// TwinCAT 3 PLC project PLCStudent
// ProgramVersion: 3.1.4022.4
// libraries:
//   Tc2_Standard, * (Beckhoff Automation GmbH)
//   Tc2_System, * (Beckhoff Automation GmbH)
//   Tc3_Module, * (Beckhoff Automation GmbH)
//   VisuSymbols,3.5.10.0,System
// project tree:
//   / GlobalTextList.TcGTLO, PlcTask.TcTTO (not stored), Visualization Manager.TcVMO (not stored)
//   GVLs/ GVL.TcGVL
//   POUs/ Control_AGV_SFC.TcPOU, Display_Pos.TcPOU, MAIN.TcPOU
//   VISUs/ Control_HMI.TcVIS
// (motion and I/O tree: see PLC project plcsim)
// real-time tasks:
//   TASK PlcTask: cycle T#20ms, priority 20, ADS port 350
// variable links:
//   PLCSim/PLCSim Instance <-> PLCStudent/PLCStudent Instance
//     PlcTask Inputs/GVL.iiGotoPos <-> PlcTask Outputs/GVL.qiGotoPos
//     PlcTask Inputs/GVL.ixPLCStrobe <-> PlcTask Outputs/GVL.qxPLCStrobe
//     PlcTask Outputs/GVL.qiAtPos <-> PlcTask Inputs/GVL.iiAtPos
//     PlcTask Outputs/GVL.qxAGVStrobe <-> PlcTask Inputs/GVL.ixAGVStrobe

// ---- GVLs/GVL.TcGVL
{attribute 'qualified_only'}
VAR_GLOBAL
//Input to PLC from process
	ixAGVStrobe		AT %I*:	BOOL;	(* AGV strobe signal *)
	iiAtPos			AT %I*:	INT;	(* Actual position of AGV *)
	
//Output from PLC to process
	qxPLCStrobe		AT %Q*:	BOOL;	(* PLC strobe signal *)
	qiGotoPos		AT %Q*:	INT;	(* Target position for AGV *)
	
	sTargetList : ARRAY [1..5] OF STRING := ['HOME','A', 'B', 'C', 'D'];
	Position : INT:=0;
	ixStartButton : BOOL;
	ixStopButton : BOOL;
	ixResetButton : BOOL;
	qxDIsplay_Pos : STRING;
	qxReadylamp : BOOL;
	qxMovinglamp : BOOL;
	qxStoplamp : BOOL;
	qxStopEvent : BOOL;
END_VAR

// ---- POUs/Control_AGV_SFC.TcPOU
PROGRAM Control_AGV_SFC
VAR
END_VAR

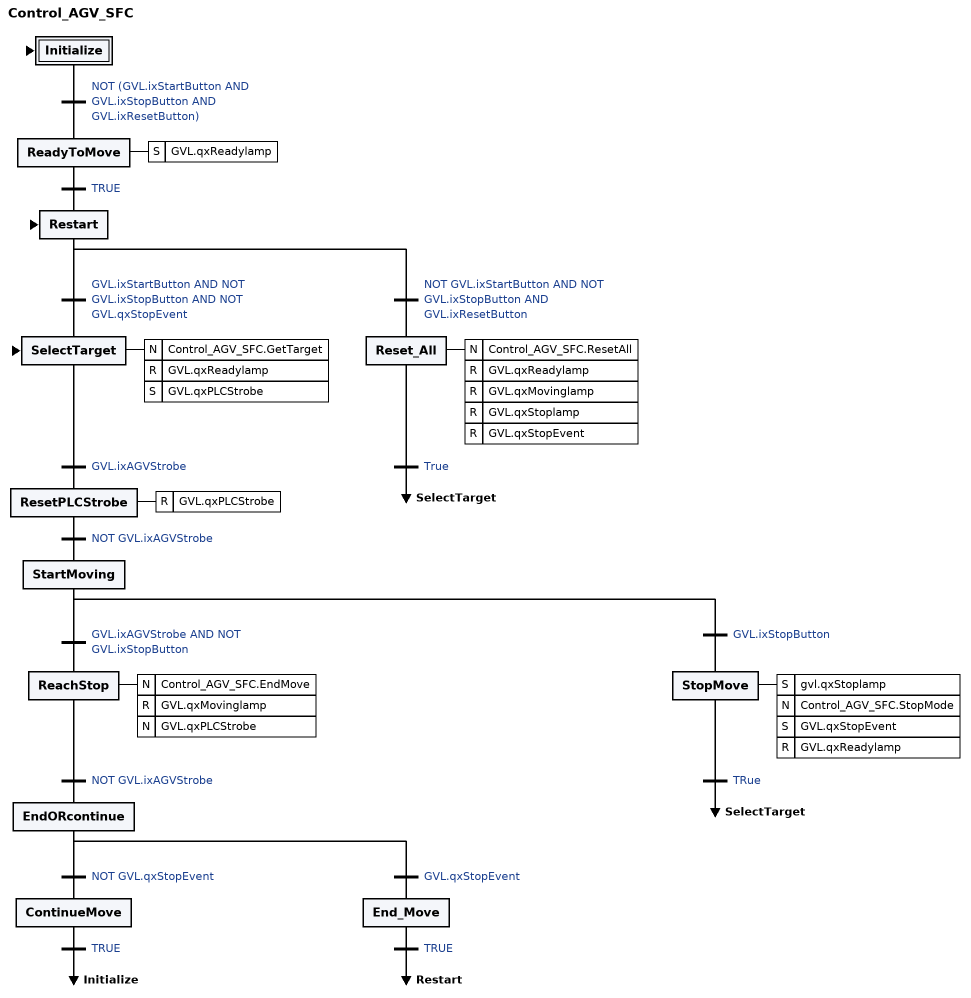
INITIAL_STEP Initialize:
END_STEP
TRANSITION FROM Initialize TO ReadyToMove
    := NOT (GVL.ixStartButton AND GVL.ixStopButton AND GVL.ixResetButton);
END_TRANSITION
STEP ReadyToMove:
    GVL.qxReadylamp(S);
END_STEP
TRANSITION FROM ReadyToMove TO Restart
    := TRUE;
END_TRANSITION
STEP Restart:
END_STEP
TRANSITION FROM Restart TO SelectTarget
    := GVL.ixStartButton AND NOT GVL.ixStopButton AND NOT GVL.qxStopEvent;
END_TRANSITION
STEP SelectTarget:
    Control_AGV_SFC.GetTarget(N);
    GVL.qxReadylamp(R);
    GVL.qxPLCStrobe(S);
END_STEP
TRANSITION FROM SelectTarget TO ResetPLCStrobe
    := GVL.ixAGVStrobe;
END_TRANSITION
STEP ResetPLCStrobe:
    GVL.qxPLCStrobe(R);
END_STEP
TRANSITION FROM ResetPLCStrobe TO StartMoving
    := NOT GVL.ixAGVStrobe;
END_TRANSITION
STEP StartMoving:
END_STEP
TRANSITION FROM StartMoving TO ReachStop
    := GVL.ixAGVStrobe AND NOT GVL.ixStopButton;
END_TRANSITION
TRANSITION FROM StartMoving TO StopMove
    := GVL.ixStopButton;
END_TRANSITION
STEP StopMove:
    gvl.qxStoplamp(S);
    Control_AGV_SFC.StopMode(N);
    GVL.qxStopEvent(S);
    GVL.qxReadylamp(R);
END_STEP
TRANSITION FROM StopMove TO SelectTarget
    := TRue;
END_TRANSITION
STEP ReachStop:
    Control_AGV_SFC.EndMove(N);
    GVL.qxMovinglamp(R);
    GVL.qxPLCStrobe(N);
END_STEP
TRANSITION FROM ReachStop TO EndORcontinue
    := NOT GVL.ixAGVStrobe;
END_TRANSITION
STEP EndORcontinue:
END_STEP
TRANSITION FROM EndORcontinue TO ContinueMove
    := NOT GVL.qxStopEvent;
END_TRANSITION
STEP ContinueMove:
END_STEP
TRANSITION FROM ContinueMove TO Initialize
    := TRUE;
END_TRANSITION
TRANSITION FROM EndORcontinue TO End_Move
    := GVL.qxStopEvent;
END_TRANSITION
STEP End_Move:
END_STEP
TRANSITION FROM End_Move TO Restart
    := TRUE;
END_TRANSITION
TRANSITION FROM Restart TO Reset_All
    := NOT GVL.ixStartButton AND NOT GVL.ixStopButton AND GVL.ixResetButton;
END_TRANSITION
STEP Reset_All:
    Control_AGV_SFC.ResetAll(N);
    GVL.qxReadylamp(R);
    GVL.qxMovinglamp(R);
    GVL.qxStoplamp(R);
    GVL.qxStopEvent(R);
END_STEP
TRANSITION FROM Reset_All TO SelectTarget
    := True;
END_TRANSITION

ACTION EndMove:
GVL.qiGotoPos:= 0;
END_ACTION

ACTION GetTarget:
GVL.qiGotoPos:= GVL.Position;
END_ACTION

ACTION ResetAll:
GVL.qiGotoPos:=1;
END_ACTION

ACTION StopMode:
GVL.qiGotoPos:= 6;
END_ACTION

END_PROGRAM

// ---- POUs/Display_Pos.TcPOU
PROGRAM Display_Pos
VAR
END_VAR

IF GVL.iiAtPos = 1 THEN
	GVL.qxDIsplay_Pos := 'HOME';
ELSIF GVL.iiAtPos = 2 THEN
	GVL.qxDIsplay_Pos := 'A';
ELSIF GVL.iiAtPos = 3 THEN
	GVL.qxDIsplay_Pos := 'B';
ELSIF GVL.iiAtPos = 4 THEN
	GVL.qxDIsplay_Pos := 'C';
ELSIF GVL.iiAtPos = 5 THEN
	GVL.qxDIsplay_Pos := 'D';
ELSIF GVL.iiAtPos = 6 THEN
	GVL.qxDIsplay_Pos := 'STOP AGV';
END_IF

END_PROGRAM

// ---- POUs/MAIN.TcPOU
PROGRAM MAIN
VAR
	
END_VAR

Control_AGV_SFC();
Display_Pos();

END_PROGRAM

// ---- GlobalTextList.TcGTLO
TEXTLIST GlobalTextList
  737 = '%s'
  90 = 'Display Position'
  274 = 'Moving'
  820 = 'Ready'
  125 = 'Reset'
  781 = 'Select Target'
  672 = 'Start'
  696 = 'Stop'
  758 = 'Stopped'
  217 = 'Target Position'
END_TEXTLIST

// ---- VISUs/Control_HMI.TcVIS
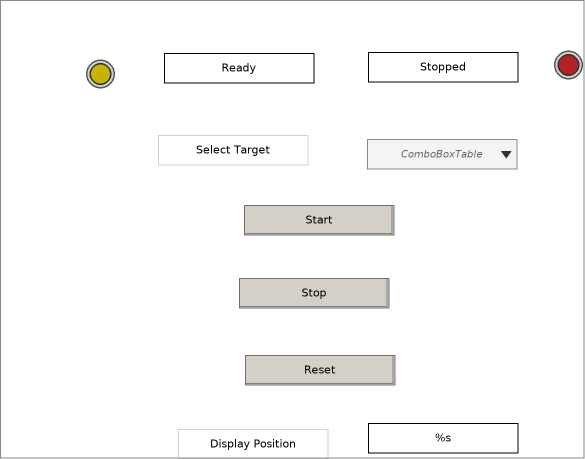
VISUALIZATION Control_HMI  // 585x459
    Textfield (158,135 150x30), "Select Target"
    Rectangle (368,423 150x30), "%s", text variable: GVL.qxDIsplay_Pos
    Textfield (178,429 150x30), "Display Position"
    Button (244,205 150x30), "Start"
        tap GVL.ixStartButton
    Button (239,278 150x30), "Stop"
        tap GVL.ixStopButton
    Button (245,355 150x30), "Reset"
        tap GVL.ixResetButton
    Lamp1 (84,57 33x34), variable: GVL.qxReadylamp, style: Lamp-Lamp1-Yellow
    Lamp1 (552,48 33x34), variable: GVL.qxStoplamp, style: Lamp-Lamp1-Red
    ComboBoxTable (367,139 150x30), variable: GVL.Position, data array: GVL.sTargetList
        p3854506369: GVL.sTargetList[INDEX]
    RoundedRectangle (164,53 150x30), "Ready"
    RoundedRectangle (368,52 150x30), "Stopped"
END_VISUALIZATION
